// TwinCAT 3 PLC project Testing
// ProgramVersion: 3.1.4022.3
// libraries:
//   SysTimeRtc, * (System)
//   Tc2_MC2, * (Beckhoff Automation GmbH)
//   Tc2_NC, * (Beckhoff Automation GmbH)
//   Tc2_Standard, * (Beckhoff Automation GmbH)
//   Tc2_System, * (Beckhoff Automation GmbH)
//   Tc2_Utilities, * (Beckhoff Automation GmbH)
//   Tc3_MC2_AdvancedHoming, * (Beckhoff Automation GmbH)
//   Tc3_Module, * (Beckhoff Automation GmbH)
//   VisuDialogs, * (System)
// project tree:
//   DUTs/ E_LED_Errors.TcDUT, E_LED_State.TcDUT, ST_LEDSystem.TcDUT, ST_LED.TcDUT, ST_Log.TcDUT, ST_Request.TcDUT
//   / GlobalTextList.TcGTLO, PlcTask.TcTTO, Visualization Manager.TcVMO (not stored), VISU_TASK.TcTTO
//   GVLs/ EMPTY.TcGVL
//   POUs/ AddRequest.TcPOU, F_WRITE_LOG.TcPOU, F_WRITE_MEMORY.TcPOU, MAIN.TcPOU, TimeReceive.TcPOU, TriggerCurrentTime.TcPOU
//   VISUs/ Visualization.TcVIS
// real-time tasks:
//   TASK PlcTask: cycle T#10ms, priority 20, ADS port 350
//   TASK VISU_TASK: cycle T#200000us, priority 30, ADS port 351
// motion (NC):
//   TASK NC-Task 1 SAF: cycle T#2ms, priority 4, ADS port 501
//   TASK NC-Task 1 SVB: cycle T#10ms, priority 8, ADS port 511
//   AXIS Axis A (id 1)
//     OtherSettings: AllowMotionCmdToSlave=true
//     encoder EncType=1
//     drive DrvType=5
//       Analog: ScaleFactorActTorque=0.1
//       TimeComp: TaskDelayCycles=1
//     controller CtrType=1
//       CtrPara: PriorControlFactor=1
//         Observer: BandWidth=20
//   AXIS Axis B (id 2)
//     OtherSettings: AllowMotionCmdToSlave=true
//     encoder EncType=1
//     drive DrvType=5
//       Analog: ScaleFactorActTorque=0.1
//       TimeComp: TaskDelayCycles=1
//     controller CtrType=1
//       CtrPara: PriorControlFactor=1
//         Observer: BandWidth=20
// I/O:
//   DEVICE Device 1 (EtherCAT), AmsNetId 10.160.29.112.2.1

CONFIGURATION Testing
    RESOURCE PLC ON TwinCAT3
        TASK PlcTask(INTERVAL := T#10ms, PRIORITY := 20);
        TASK VISU_TASK(INTERVAL := T#200000us, PRIORITY := 30);
        PROGRAM MAIN WITH PlcTask : MAIN;
        PROGRAM VisuElems_Visu_Prg WITH VISU_TASK : VisuElems.Visu_Prg;
    END_RESOURCE
END_CONFIGURATION

// ---- DUTs/E_LED_Errors.TcDUT
{attribute 'qualified_only'}
{attribute 'strict'}
TYPE E_LED_Errors :
(
	disconnected := 0,
	none := 1
);
END_TYPE

// ---- DUTs/E_LED_State.TcDUT
{attribute 'qualified_only'}
{attribute 'strict'}
TYPE E_LED_State :
(
	disabled := 0,
	enabled := 1,
	finished := 2	
);
END_TYPE

// ---- DUTs/ST_LEDSystem.TcDUT
TYPE ST_LEDSystem :
STRUCT
	stLED_r: ST_LED := (color:='RED');
	stLED_o: ST_LED := (color:='ORANGE');
	stLED_g: ST_LED := (color:='GREEN');
	arrLog: ARRAY [0..100] OF ST_Log;
	stRequest_r: ST_Request := ();
	stRequest_o: ST_Request := ();
	stRequest_g: ST_Request := ();
	stProcessing_r: ST_Request := ();
	stProcessing_o: ST_Request := ();
	stProcessing_g: ST_Request := ();
END_STRUCT
END_TYPE

// ---- DUTs/ST_LED.TcDUT
TYPE ST_LED :
STRUCT
	eLEDState: E_LED_STATE;
	eLEDErrorStatus: E_LED_Errors;
	bRequestApproved: BOOL;
	fbTimer: TON := (IN:=FALSE);
	fbTrigger: R_TRIG := (CLK:=fbTimer.Q);
	tTarget: TIME;
	color: STRING;
END_STRUCT
END_TYPE

// ---- DUTs/ST_Log.TcDUT
TYPE ST_Log :
STRUCT
	sTime: DT;
	sStatus: STRING;
END_STRUCT
END_TYPE

// ---- DUTs/ST_Request.TcDUT
TYPE ST_Request :
STRUCT
	stTargetLED: ST_LED;
	tTargetTime: TIME;
	exists: BOOL := FALSE;
END_STRUCT
END_TYPE

// ---- GVLs/EMPTY.TcGVL
{attribute 'qualified_only'}
VAR_GLOBAL
	stEmptyRequest: ST_Request := ();
	sEmptyString: STRING := '';
	tTime: DT;
END_VAR

// ---- POUs/MAIN.TcPOU
PROGRAM MAIN
(*	- Project: My Light Status: A Documented Study OF PLC State Machines
		- execution process:
			1. UI Pops up, with both light modules showing up
			2. Job is to click through the lights using the mouse. Whichever ones are "turned on" will the be packaged as a request file:
				- when the "submit request" has button has been clicked on
				- time is fixable, if it isn't fixed, it will be set to 3 seconds
				- if there is no assignment added to the stack, the LED will shut off
			3. Output:
				- edited physical LED state, reflects the UI
				- update log
					- previous color
					- time elapsed for the light state(current, then move it to the log)
				- blanks out the LED when there's no requests going no
*)
VAR
	print: STRING := '';
	fbTimerRed: TON;
	fbTimerOrange: TON;
	fbTimerGreen: TON;
	stSystem : ST_LEDSystem; //creation of the entire system structure, see ST_LEDSystem in DUT
	//reader variables
	sUserRequestInput_r: STRING := EMPTY.sEmptyString;
	sUserRequestInput_o: STRING := EMPTY.sEmptyString;
	sUserRequestInput_g: STRING := EMPTY.sEmptyString;	
END_VAR

EMPTY.tTime := TimeReceive();

fbTimerRed(IN:=stSystem.stProcessing_r.exists, PT:=stSystem.stProcessing_r.tTargetTime);
fbTimerOrange(IN:=stSystem.stProcessing_o.exists, PT:=stSystem.stProcessing_o.tTargetTime);
fbTimerGreen(IN:=stSystem.stProcessing_g.exists, PT:=stSystem.stProcessing_g.tTargetTime);

IF(stSystem.stLED_r.eLEDState = E_LED_State.disabled AND stSystem.stRequest_r.exists) THEN
	stSystem.stProcessing_r := stSystem.stRequest_r;
	stSystem.stRequest_r := EMPTY.stEmptyRequest;
	F_WRITE_LOG(inputColor:=stSystem.stLED_r,status:='color processed');
END_IF

IF(stSystem.stLED_o.eLEDState = E_LED_State.disabled AND stSystem.stRequest_o.exists) THEN
	stSystem.stProcessing_o := stSystem.stRequest_o;
	stSystem.stRequest_o := EMPTY.stEmptyRequest;
	F_WRITE_LOG(inputColor:=stSystem.stLED_o,status:='color processed');
END_IF

IF(stSystem.stLED_g.eLEDState = E_LED_State.disabled AND stSystem.stRequest_g.exists) THEN
	stSystem.stProcessing_g := stSystem.stRequest_g;
	stSystem.stRequest_g := EMPTY.stEmptyRequest;
	F_WRITE_LOG(inputColor:=stSystem.stLED_g,status:='color processed');
END_IF

IF(fbTimerGreen.IN) THEN
	stSystem.stLED_g.eLEDState := E_LED_State.enabled;
END_IF

IF(fbTimerOrange.IN) THEN
	stSystem.stLED_o.eLEDState := E_LED_State.enabled;
END_IF

IF(fbTimerRed.IN) THEN
	stSystem.stLED_r.eLEDState := E_LED_State.enabled;
END_IF

IF(fbTimerGreen.Q) THEN
	stSystem.stLED_g.eLEDState := E_LED_State.disabled;
	stSystem.stProcessing_g := EMPTY.stEmptyRequest;
	F_WRITE_LOG(inputColor:=stSystem.stLED_g,status:='process complete');
END_IF

IF(fbTimerOrange.Q) THEN
	stSystem.stLED_o.eLEDState := E_LED_State.disabled;
	stSystem.stProcessing_o := EMPTY.stEmptyRequest;
	F_WRITE_LOG(inputColor:=stSystem.stLED_o,status:='process complete');
END_IF

IF(fbTimerRed.Q) THEN
	stSystem.stLED_r.eLEDState := E_LED_State.disabled;
	stSystem.stProcessing_r := EMPTY.stEmptyRequest;
	F_WRITE_LOG(inputColor:=stSystem.stLED_r,status:='process complete');
END_IF

END_PROGRAM

// ---- POUs/TimeReceive.TcPOU
FUNCTION TimeReceive
VAR
Date_and_time_in_seconds	: UDINT;
Local_date_time_seconds	: UDINT;
Date_and_Time_result	: UDINT;
Local_date_time_from_secs	: SYSTIMEDATE;
Date_and_time_string	: STRING;
Err_result: UDINT;
END_VAR
VAR_OUTPUT
Date_and_time_format	: DATE_AND_TIME;
END_VAR

// Get time in seconds since 1970 :
Date_and_time_in_seconds := SysTimeRtcGet(Err_result);
IF Date_and_Time_result <> 0 THEN
RETURN;
END_IF

// Convert UTC seconds to local time seconds, regarding Timezone and Summer time :
Date_and_Time_result := SysTimeRtcConvertUtcToLocal(Date_and_time_in_seconds, Local_date_time_seconds);
IF Date_and_Time_result <> 0 THEN
RETURN;
END_IF

// Convert the UTC seconds to a DATE_AND_TIME variable dt#yyyy-mm-dd-hh:mm:ss :
Date_and_time_format := UDINT_TO_DT(Local_date_time_seconds);
RETURN;

// Convert DATE_AND_TIME to a String :
Date_and_time_string := DT_TO_STRING(Date_and_time_format);

END_FUNCTION

// ---- POUs/F_WRITE_LOG.TcPOU
FUNCTION F_WRITE_LOG : BOOL
VAR_INPUT
	inputColor: ST_LED; 
	status: STRING;
END_VAR
VAR
	stLOG: ST_Log := (sStatus:=CONCAT(CONCAT(status, ' -'), inputColor.color)); //log to be added to the log collection
END_VAR

stLog.sTime := EMPTY.tTime;
F_WRITE_MEMORY(cbData:=SIZEOF(stLog),pData:=ADR(stLog),cbBuffer:=SIZEOF(MAIN.stSystem.arrLog),pBuffer:=ADR(MAIN.stSystem.arrLog));

END_FUNCTION

// ---- POUs/F_WRITE_MEMORY.TcPOU
FUNCTION F_WRITE_MEMORY : BOOL
VAR_INPUT
	cbData : UDINT;
	pData : POINTER TO BYTE;
	cbBuffer : UDINT;
	pBuffer : POINTER TO BYTE;
END_VAR
VAR
END_VAR

FW_MemMove(pDest:=pBuffer + cbData,pSrc:=pBuffer,cbLen:=cbBuffer-cbData);

FW_MemMove(pDest:=pBuffer,pSrc:=pData,cbLen:=cbData);

END_FUNCTION

// ---- POUs/AddRequest.TcPOU
FUNCTION AddRequest : BOOL
VAR_INPUT
	
END_VAR
VAR
END_VAR
VAR_OUTPUT
	bFinishStatus: BOOL;
END_VAR

END_FUNCTION

// ---- POUs/TriggerCurrentTime.TcPOU
FUNCTION TriggerCurrentTime : BOOL
VAR_INPUT
END_VAR
VAR
END_VAR
VAR_OUTPUT
	returner: BOOL;
END_VAR


RETURN;

END_FUNCTION

// ---- GlobalTextList.TcGTLO
TEXTLIST GlobalTextList
  448 = '\tRed'
  730 = '     Orange'
  982 = '    Green'
  669 = '    Orange'
  881 = '    Red'
  118 = '%d'
  571 = '%s'
  506 = '+'
  197 = 'Elapsed: '
  84 = 'Elapsed: %d'
  774 = 'Elapsed: %s'
  133 = 'Graphical Representation of LED Request System and Status'
  797 = 'Greee'
  353 = 'Green'
  221 = 'MAIN.stSystem.arrLog[INDEX].sStatus'
  677 = 'Make red request'
  973 = 'Make Requests'
  533 = 'Orange'
  377 = 'Red'
  593 = 'Request Stack'
  638 = 'Request Stack:'
  738 = 'String value: %s'
  433 = 'String value: %s, Double value:%d'
  154 = 'StructuresTest.'
  407 = 't#3s'
END_TEXTLIST

// ---- VISUs/Visualization.TcVIS
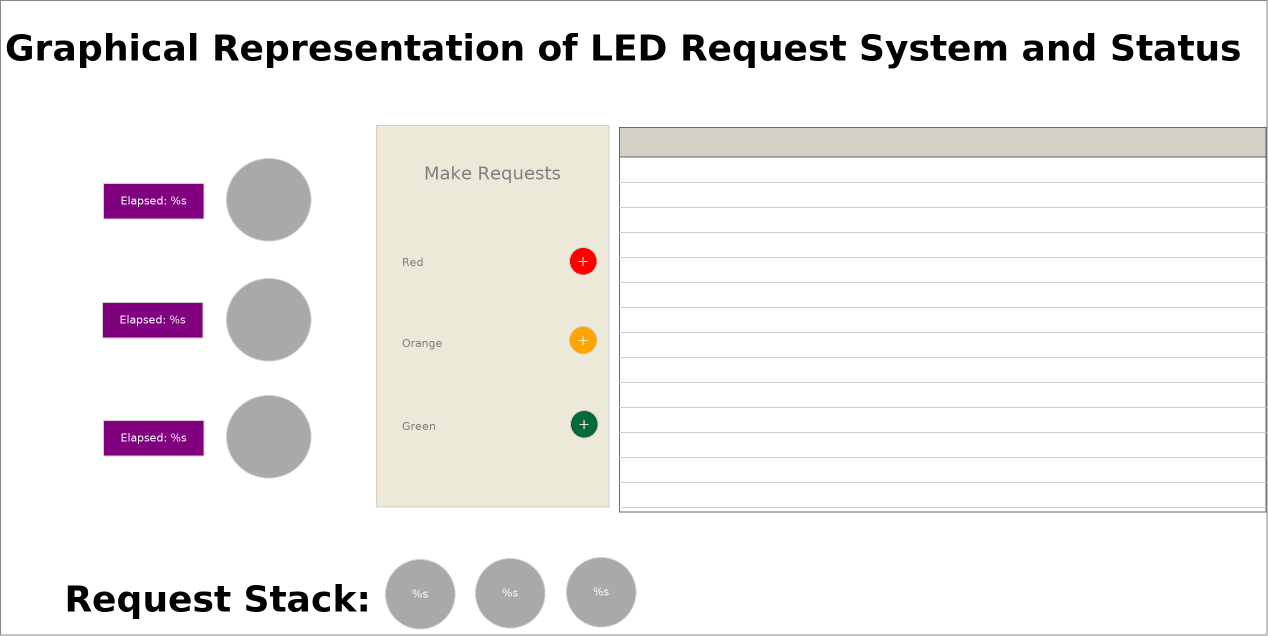
VISUALIZATION Visualization  // 1268x636
    Label (9,13 1229x70), "Graphical Representation of LED Request System and Status"
    Ellipse (226,158 85x83), colour toggle: MAIN.stSystem.stLED_r.eLEDState = E_LED_State.enabled
    Ellipse (226,278 85x83), colour toggle: MAIN.stSystem.stLED_o.eLEDState = E_LED_State.enabled
    Ellipse (226,395 85x83), colour toggle: MAIN.stSystem.stLED_g.eLEDState = E_LED_State.enabled
    Rectangle (103,183 101x36), "Elapsed: %s", text variable: MAIN.fbTimerRed.ET
    Rectangle (103,420 101x36), "Elapsed: %s", text variable: MAIN.fbTimerGreen.ET
    Rectangle (102,302 101x36), "Elapsed: %s", text variable: MAIN.fbTimerOrange.ET
    Label (39,564 358x70), "Request Stack:"
    Ellipse (385,559 70x70), "%s", text variable: time_to_string(MAIN.stSystem.stRequest_r.tTargetTime), colour toggle: MAIN.stSystem.stRequest_r.exists
    Ellipse (475,558 70x70), "%s", text variable: time_to_string(MAIN.stSystem.stRequest_o.tTargetTime), colour toggle: MAIN.stSystem.stRequest_o.exists
    Ellipse (566,557 70x70), "%s", text variable: time_to_string(MAIN.stSystem.stRequest_g.tTargetTime), colour toggle: MAIN.stSystem.stRequest_g.exists
    Rectangle (376,125 233x382)
    Rectangle (381,153 223x41), "Make Requests"
    Rectangle (385,244 176x37), "Red"
    Rectangle (385,325 176x37), "Orange"
    Rectangle (385,408 176x37), "Green"
    Ellipse (569,247 28x28), "+", colour toggle: MAIN.stSystem.stRequest_r.exists
        OnMouseDown: execute {
            IF(MAIN.stSystem.stRequest_r.exists = FALSE) THEN
            	IF len(Main.sUserRequestInput_r) = 0 THEN
            		Main.stSystem.stRequest_r.tTargetTime := T#3S;
            	ELSE
            		Main.stSystem.stRequest_r.tTargetTime := STRING_TO_TIME(Main.sUserRequestInput_r);
            	END_IF
            	MAIN.stSystem.stRequest_r.exists := TRUE;
            	MAIN.sUserRequestInput_r := EMPTY.sEmptyString;
            	F_WRITE_LOG(inputColor:=MAIN.stSystem.stLED_r,status:='request made');
            END_IF
        }
    Ellipse (569,326 28x28), "+", colour toggle: MAIN.stSystem.stRequest_o.exists
        OnMouseDown: execute {
            IF(MAIN.stSystem.stRequest_o.exists = FALSE) THEN
            	IF len(Main.sUserRequestInput_o) = 0 THEN
            		Main.stSystem.stRequest_o.tTargetTime := T#3S;
            	ELSE
            		Main.stSystem.stRequest_o.tTargetTime := STRING_TO_TIME(Main.sUserRequestInput_o);
            	END_IF
            	MAIN.stSystem.stRequest_o.exists := TRUE;
            	MAIN.sUserRequestInput_o := EMPTY.sEmptyString;
            	F_WRITE_LOG(inputColor:=MAIN.stSystem.stLED_o,status:='request made');
            END_IF
        }
    Textfield (432,247 126x30)
        OnMouseDown: write MAIN.sUserRequestInput_r via Edit
    Textfield (447,327 111x30)
        OnMouseDown: write MAIN.sUserRequestInput_o via Edit
    Textfield (441,411 117x30)
        OnMouseDown: write MAIN.sUserRequestInput_g via InputWithLimits
    Ellipse (570,410 28x28), "+", colour toggle: MAIN.stSystem.stRequest_g.exists
        OnMouseDown: execute {
            IF(MAIN.stSystem.stRequest_g.exists = FALSE) THEN
            	IF len(Main.sUserRequestInput_g) = 0 THEN
            		Main.stSystem.stRequest_g.tTargetTime := T#3S;
            	ELSE
            		Main.stSystem.stRequest_g.tTargetTime := STRING_TO_TIME(Main.sUserRequestInput_g);
            	END_IF
            	MAIN.stSystem.stRequest_g.exists := TRUE;
            	MAIN.sUserRequestInput_g := EMPTY.sEmptyString;
            	F_WRITE_LOG(inputColor:=MAIN.stSystem.stLED_g,status:='request made');
            END_IF
        }
    Table (619,127 647x385), data array: MAIN.stSystem.arrLog
        p3854506369: MAIN.stSystem.arrLog[INDEX].sTime
        p1892666644: MAIN.stSystem.arrLog[INDEX].sStatus
END_VISUALIZATION
